Staubli VAL3: ros_server.pjx

--- ros_server.pjx ---
Parameters version=s8.10.3Cs9_BS2093 stackSize=5000 millimeterUnit=true
Program file=dataReceiver.pgx
Program file=dataReceiverIO.pgx
Program file=dataStreamer.pgx
Program file=decodeMsgBody.pgx
Program file=decodeMsgBodyIO.pgx
Program file=decodeMsgHeader.pgx
Program file=decodeMsgHeaderIO.pgx
Program file=decTrajPt.pgx
Program file=decTrajPtFull.pgx
Program file=encodeAck.pgx
Program file=encodeAckIO.pgx
Program file=encodeJState.pgx
Program file=encodeStatus.pgx
Program file=encPrefixHeader.pgx
Program file=encTrajPtAck.pgx
Program file=encTrajPtFAck.pgx
Program file=fetchStatus.pgx
Program file=handleRequest.pgx
Program file=initParams.pgx
Program file=initRosMsg.pgx
Program file=interpolateVel.pgx
Program file=motionControl.pgx
Program file=pushMotion.pgx
Program file=pushMotionIO.pgx
Program file=recvData.pgx
Program file=recvHeartbeat.pgx
Program file=recvMsgBody.pgx
Program file=recvMsgBodyIO.pgx
Program file=recvMsgHeader.pgx
Program file=recvMsgHeaderIO.pgx
Program file=recvRosMsg.pgx
Program file=recvTrajPt.pgx
Program file=recvTrajPtFull.pgx
Program file=screenUpdate.pgx
Program file=sendAck.pgx
Program file=sendAckIO.pgx
Program file=sendData.pgx
Program file=sendRosMsg.pgx
Program file=setupRosMsgs.pgx
Program file=start.pgx
Program file=stop.pgx
Program file=toJointArrayRad.pgx
Program file=toJointRxDeg.pgx
Data file=ros_server.dtx
Library alias=libQueueFuncs path=Disk://ros_libs/QueueFuncs/QueueFuncs.pjx
Library alias=libInterface path=Disk://ros_libs/UserInterface/interfaceDefault/interfaceDefault.pjx autoload=false
Library alias=Staubli path=Disk://ros_libs/Staubli/Staubli.pjx
Library alias=IO path=Disk://ros_libs/IOInterface/IOInterface.pjx
Library alias=SimpleMsg path=Disk://ros_libs/SimpleMessage/SimpleMessage.pjx
Type name=RosSimpleMsg path=Disk://ros_libs/RosSimpleMsg/RosSimpleMsg.pjx
Type name=RobotStatusMsg path=Disk://ros_libs/RobotStatusMsg/RobotStatusMsg.pjx
Type name=JointStateMsg path=Disk://ros_libs/JointStateMsg/JointStateMsg.pjx
Type name=JointTrajPtMsg path=Disk://ros_libs/JointTrajPtMsg/JointTrajPtMsg.pjx
Type name=JointTrajPtFMsg path=Disk://ros_libs/JointTrajPtFMsg/JointTrajPtFMsg.pjx
Type name=JointFbkMsg path=Disk://ros_libs/JointFbkMsg/JointFbkMsg.pjx
Type name=MotionCmd path=Disk://ros_libs/MotionCmd/MotionCmd.pjx
Type name=Header path=Disk://ros_libs/Header/Header.pjx
Type name=Prefix path=Disk://ros_libs/Prefix/Prefix.pjx
Type name=Body path=Disk://ros_libs/Body/Body.pjx
Type name=Queue path=Disk://ros_libs/Queue/Queue.pjx

--- ros_server.dtx ---
public bool bFbkOverrun
public bool bMotionOverrun
public sio siTcpIpFbk = {link=Socket\Feedback}
public sio siTcpIpMotion = {link=Socket\Motion}
public string sStreamTaskName = "publisher"
public string sMotionTaskName
public RosSimpleMsg rosGenericMsg
  [0]
    Header header
      [0]
        num nMsgType
        num nCommType
        num nReplyCode
        num nData[12]
    Prefix prefix
      [0]
        num nLength
        num nData[4]
public tool tTool = {fatherId=flange[0], ioLink=ValveIO\valve1}
public string sTrajPtTaskName
public bool bTrajPtOverrun
public RobotStatusMsg rosStatusMsg
  [0]
    Body body
      [0]
        num nData[28]
    Header header
      [0]
        num nMsgType
        num nCommType
        num nReplyCode
        num nData[12]
    Prefix prefix
      [0]
        num nLength
        num nData[4]
    RobotStatus robotStatus
      [0]
        num nDrivesPowered
        num nEStopped
        num nErrorCode
        num nInError
        num nInMotion
        num nMode
        num nMotionPossible
public JointStateMsg rosJointMsg
  [0]
    Header header
      [0]
        num nMsgType
        num nCommType
        num nReplyCode
        num nData[12]
    Body body
      [0]
        num nData[44]
    JointState jointState
      [0]
        num nSeq
        num nJoints[10]
    Prefix prefix
      [0]
        num nLength
        num nData[4]
public JointTrajPtMsg rosTrajPtMsg
  [0]
    Header header
      [0]
        num nMsgType
        num nCommType
        num nReplyCode
        num nData[12]
    JointTrajPt jointTrajPt
      [0]
        num nSeq
        num nJoints[10]
        num nVelocity
        num nDuration
    Prefix prefix
      [0]
        num nLength
        num nData[4]
    Body body
      [0]
        num nData[52]
public JointTrajPtFMsg rosTrajPtFMsg
  [0]
    Header header
      [0]
        num nMsgType
        num nCommType
        num nReplyCode
        num nData[12]
    Prefix prefix
      [0]
        num nLength
        num nData[4]
    JointTrajPtFull jointTrajPtFull
      [0]
        num nRobotId
        num nSeq
        num nValidFields
        num nTime
        num nPositions[10]
        num nVelocities[10]
        num nAccelerations[10]
    Body body
      [0]
        num nData[136]
public JointFbkMsg rosJointFbkMsg
  [0]
    Header header
      [0]
        num nMsgType
        num nCommType
        num nReplyCode
        num nData[12]
    Prefix prefix
      [0]
        num nLength
        num nData[4]
    JointFeedback jointFeedback
      [0]
        num nRobotId
        num nValidFields
        num nTime
        num nPositions[10]
        num nVelocities[10]
        num nAccelerations[10]
    Body body
      [0]
        num nData[132]
public JointTrajPtFMsg rosTrajPtFAck
  [0]
    Header header
      [0]
        num nMsgType
        num nCommType
        num nReplyCode
        num nData[12]
    Prefix prefix
      [0]
        num nLength
        num nData[4]
    JointTrajPtFull jointTrajPtFull
      [0]
        num nRobotId
        num nSeq
        num nValidFields
        num nTime
        num nPositions[10]
        num nVelocities[10]
        num nAccelerations[10]
    Body body
      [0]
        num nData[136]
public JointTrajPtMsg rosTrajPtAck
  [0]
    Header header
      [0]
        num nMsgType
        num nCommType
        num nReplyCode
        num nData[12]
    JointTrajPt jointTrajPt
      [0]
        num nSeq
        num nJoints[10]
        num nVelocity
        num nDuration
    Prefix prefix
      [0]
        num nLength
        num nData[4]
    Body body
      [0]
        num nData[52]
public bool bScreenOverrun
public string sScreenTaskName
public num nInConnFlag
public num nOutConnFlag
public string sHtbtTaskName
public num nPtsPopped
public bool bStopNow
public num nMotionProgress
public num nMoveId
public num nMovePts
public num nElapsedTime
public num nHeaderTime
public bool bOverwriteVel
public Queue qMoveBuffer
  [0]
    num nPush
    num nPop
    num nElems
    MotionCmd buffer[10]
      [0]
        mdesc mDesc = {leave=0, reach=0}
        num nDuration
        num nSequence
        jointRx jJointRx
      [1]
        mdesc mDesc = {leave=0, reach=0}
        num nDuration
        num nSequence
        jointRx jJointRx
      [2]
        mdesc mDesc = {leave=0, reach=0}
        num nDuration
        num nSequence
        jointRx jJointRx
      [3]
        mdesc mDesc = {leave=0, reach=0}
        num nDuration
        num nSequence
        jointRx jJointRx
      [4]
        mdesc mDesc = {leave=0, reach=0}
        num nDuration
        num nSequence
        jointRx jJointRx
      [5]
        mdesc mDesc = {leave=0, reach=0}
        num nDuration
        num nSequence
        jointRx jJointRx
      [6]
        mdesc mDesc = {leave=0, reach=0}
        num nDuration
        num nSequence
        jointRx jJointRx
      [7]
        mdesc mDesc = {leave=0, reach=0}
        num nDuration
        num nSequence
        jointRx jJointRx
      [8]
        mdesc mDesc = {leave=0, reach=0}
        num nDuration
        num nSequence
        jointRx jJointRx
      [9]
        mdesc mDesc = {leave=0, reach=0}
        num nDuration
        num nSequence
        jointRx jJointRx
public Queue qTrajPtBuffer
  [0]
    num nPush
    num nPop
    num nElems
    MotionCmd buffer[10]
      [0]
        mdesc mDesc = {leave=0, reach=0}
        num nDuration
        num nSequence
        jointRx jJointRx
      [1]
        mdesc mDesc = {leave=0, reach=0}
        num nDuration
        num nSequence
        jointRx jJointRx
      [2]
        mdesc mDesc = {leave=0, reach=0}
        num nDuration
        num nSequence
        jointRx jJointRx
      [3]
        mdesc mDesc = {leave=0, reach=0}
        num nDuration
        num nSequence
        jointRx jJointRx
      [4]
        mdesc mDesc = {leave=0, reach=0}
        num nDuration
        num nSequence
        jointRx jJointRx
      [5]
        mdesc mDesc = {leave=0, reach=0}
        num nDuration
        num nSequence
        jointRx jJointRx
      [6]
        mdesc mDesc = {leave=0, reach=0}
        num nDuration
        num nSequence
        jointRx jJointRx
      [7]
        mdesc mDesc = {leave=0, reach=0}
        num nDuration
        num nSequence
        jointRx jJointRx
      [8]
        mdesc mDesc = {leave=0, reach=0}
        num nDuration
        num nSequence
        jointRx jJointRx
      [9]
        mdesc mDesc = {leave=0, reach=0}
        num nDuration
        num nSequence
        jointRx jJointRx
num nVel[2]
num nStdMsgType{}
  [JOINT_TRAJ_PT] = 11
  [JOINT_TRAJ_PT_FULL] = 14
  [WRITE_SINGLE_IO] = {}
num nCommType{}
  [SERVICE_REQUEST] = 2
mdesc mNomSpeed
num nRecHeader
num nDecHeader = 1
num nRecBody = 2
num nDecBody = 3
num nPushMotion = 4
num nAck = 5
num nReset
public RosSimpleMsg genericIOMsg
  [0]
    Header header
      [0]
        num nMsgType
        num nCommType
        num nReplyCode
        num nData[12]
    Prefix prefix
      [0]
        num nLength
        num nData[4]
num nConnFlagIO
public string sIORequestTaskName
num nConnFlagMotion
public sio siTcpIpIO = {link=Socket\IO}
num ntest
string sTest

--- start.pgx ---
program start()
  local num l_nFbkPeriod
  local num l_nMotionPeriod
  local num l_nTrajPeriod
  local num l_nScreenUpdate
  local string l_sVersionMajor
  local num l_nVersionMajor
  local bool l_bOkMajor
  local string l_sVersionMinor
  local num l_nVersionMinor
  local bool l_bOkMinor
begin
  // Copyright (c) 2016, Ocado Technology - Robotics Research Team
  //
  // Licensed under the Apache License, Version 2.0 (the "License");
  // you may not use this file except in compliance with the License.
  // You may obtain a copy of the License at
  //
  //     http://www.apache.org/licenses/LICENSE-2.0
  //
  // Unless required by applicable law or agreed to in writing, software
  // distributed under the License is distributed on an "AS IS" BASIS,
  // WITHOUT WARRANTIES OR CONDITIONS OF ANY KIND, either express or implied.
  // See the License for the specific language governing permissions and
  // limitations under the License.


  // Load interface library for CS8 or CS9
  //
  // CS9 handles the UI differently than CS8, requires
  // the UI funtions to be loaded in seperate libraries

  if(mid(getVersion("System"),1,1) == "7")
    // CS8 - VAL 3 rev 7
    // Check for VAL 3 version >= 7.7
    l_sVersionMajor = mid(getVersion("VAL3"),1,1)
    l_sVersionMinor = mid(getVersion("VAL3"),2,1)
    toNum(l_sVersionMajor, l_nVersionMajor, l_bOkMajor)
    toNum(l_sVersionMinor, l_nVersionMinor, l_bOkMinor)
    if(!l_bOkMajor or !l_bOkMinor)
      popUpMsg("Error reading VAL 3 version")
      taskKill("ros_server~")
    endIf
    if( !((l_nVersionMajor == 7) and (l_nVersionMinor >= 7)))
      // VAL 3 version is too old
      popUpMsg("Error: VAL 3 version is < 7.7, socket communication will not work!")
      taskKill("ros_server~")
    endIf
    libInterface:libLoad("ros_libs/UserInterface/interfaceCS8")
  elseIf(mid(getVersion("System"),1,1) == "8")
    // CS9 - VAL 3 rev 8
    libInterface:libLoad("ros_libs/UserInterface/interfaceCS9")
  endIf

  // feedback task will run every 20ms (50Hz)
  l_nFbkPeriod=0.02
  //l_nFbkPeriod = 0.032 // 30Hz
  //l_nFbkPeriod = 0.05  // 20Hz
  //l_nFbkPeriod = 1.0   //  1Hz

  // motion control task will run every 4ms (250Hz)
  l_nMotionPeriod = 0.004
  //l_nMotionPeriod=0.012  // 83Hz
  //l_nMotionPeriod = 0.05 // 20Hz

  // data (trajectory) reception task will run every 4ms (250Hz)
  l_nTrajPeriod = 0.004
  // not in use at the moment
  l_nScreenUpdate = 1.0

  sStreamTaskName = "streamerTask"
  sTrajPtTaskName = "trajPtTask"
  sMotionTaskName = "motionTask"
  sIORequestTaskName = "ioRequestTask"
  sScreenTaskName = "screenTask"
  sHtbtTaskName = "htbtTask"

  // initialise TCP/IP parameters
  call initParams()

  // initialise libraries
  call SimpleMsg:init()
  call Staubli:init()
  call IO:init()
  // setup prefix and header of ROS messages
  call setupRosMsgs()

  // socket connection status flags: initially disconnected
  nConnFlagIO = 0
  nInConnFlag = 0
  nOutConnFlag = 0
  nConnFlagMotion = 0

  // flag defining whether velocity to be overwritten to max. vel.
  bOverwriteVel = false

  nPtsPopped = 0
  nMovePts = 0

  // flush buffer of incoming socket
  clearBuffer(siTcpIpIO)
  clearBuffer(siTcpIpMotion)
  // flush buffer of outgoing socket
  clearBuffer(siTcpIpFbk)

  // check if robot is not in emergency stop and wait until estop is reset
  if(esStatus() == 2)
    popUpMsg("Please reset E-Stop")
    wait(esStatus() < 2)
  endIf

  // before anything else, enable power (only works if robot is in remote mode)
  if(!isPowered())
    if(workingMode() >= 4)
      do
        enablePower()
        delay(2)
      until isPowered()
    else
      popUpMsg("Power must be enabled manually")
    endIf
  endIf

  // reset motion, potentially setting a start joint position for calling autoConnect() in the future
  resetMotion()

  // create joint state and robot status streamer task to send data to industrial_robot_client
  taskCreateSync sStreamTaskName, l_nFbkPeriod, bFbkOverrun, dataStreamer()

  // create trajectory point task to receive data from industrial_robot_client
  taskCreateSync sTrajPtTaskName, l_nTrajPeriod, bTrajPtOverrun, dataReceiver()
  //taskCreate sTrajPtTaskName, 100, dataReceiver()

  // create motion task to synchronously apply motion commands to robot
  taskCreateSync sMotionTaskName, l_nMotionPeriod, bMotionOverrun, motionControl()

  // create asynchronous task to handle io requests
  taskCreate sIORequestTaskName, 100, dataReceiverIO(siTcpIpIO, nConnFlagIO, genericIOMsg)

  // create synchronous task to update screen
  //taskCreateSync sScreenTaskName, l_nScreenUpdate, bScreenOverrun, screenUpdate()
  taskCreate sScreenTaskName, 10, screenUpdate()

  // create asynchronous task to receive heartbeat on port 11002
  taskCreate sHtbtTaskName, 10, recvHeartbeat()

end

--- dataReceiver.pgx ---
program dataReceiver()
  local num l_nMsgRecvState
  local num l_nStartTime
begin
  // Copyright (c) 2016, Ocado Technology - Robotics Research Team
  //
  // Licensed under the Apache License, Version 2.0 (the "License");
  // you may not use this file except in compliance with the License.
  // You may obtain a copy of the License at
  //
  //     http://www.apache.org/licenses/LICENSE-2.0
  //
  // Unless required by applicable law or agreed to in writing, software
  // distributed under the License is distributed on an "AS IS" BASIS,
  // WITHOUT WARRANTIES OR CONDITIONS OF ANY KIND, either express or implied.
  // See the License for the specific language governing permissions and
  // limitations under the License.



  // state machine at initial state
  // 0: receive header
  // 1: decode header
  // 2: receive body
  // 3: decode body
  // 4: push motion into buffer
  // 5: send ACK

  // Set variable constants to make sure they were not changed
  nReset=0
  nRecHeader=0
  nDecHeader=1
  nRecBody=2
  nDecBody=3
  nPushMotion=4
  nAck=5

  l_nMsgRecvState=nRecHeader
while (true)
    // usually for state machines a switch-case statement is a neat implementation
    // HOWEVER, at every iteration of while() this task is sequenced and only called
    // after whatever ms is was defined when created.
    // As a result, receiving one single message, pushing motion and sending ACK
    // would take 6 * task period using switch-case statement.
    // The desirable behaviour is to receive and decode a full message, push motion
    // into buffer and then send ACK to client WITHIN ONE ITERATION of while(),
    // hence the if statement sequence below
    l_nStartTime=clock()
    if (l_nMsgRecvState==nRecHeader)
      call recvMsgHeader(l_nMsgRecvState)
    endIf
    nHeaderTime=clock()-l_nStartTime
    if (l_nMsgRecvState==nDecHeader)
      call decodeMsgHeader(l_nMsgRecvState)
    endIf
    if (l_nMsgRecvState==nRecBody)
      call recvMsgBody(l_nMsgRecvState)
    endIf
    if (l_nMsgRecvState==nDecBody)
      call decodeMsgBody(l_nMsgRecvState)
    endIf
    if (l_nMsgRecvState==nPushMotion)
      call pushMotion(l_nMsgRecvState)
    endIf
    if (l_nMsgRecvState==nAck)
      call encodeAck()
      call sendAck(l_nMsgRecvState)
    endIf
    nElapsedTime=clock()-l_nStartTime-nHeaderTime

    // assert state machine is working OK
    if (l_nMsgRecvState<nRecHeader or l_nMsgRecvState>nAck)
      popUpMsg("Data reception state machine error")
    endIf

    // sequence task
    delay(0)


  endWhile
end

--- dataReceiverIO.pgx ---
public program dataReceiverIO(sio& x_sSocket, num& x_nConnFlag, RosSimpleMsg& x_rMsg)
  local num l_nStartTime
  local num l_nMsgRecvState
begin
  // Copyright (c) 2016, Ocado Technology - Robotics Research Team
  //
  // Licensed under the Apache License, Version 2.0 (the "License");
  // you may not use this file except in compliance with the License.
  // You may obtain a copy of the License at
  //
  //     http://www.apache.org/licenses/LICENSE-2.0
  //
  // Unless required by applicable law or agreed to in writing, software
  // distributed under the License is distributed on an "AS IS" BASIS,
  // WITHOUT WARRANTIES OR CONDITIONS OF ANY KIND, either express or implied.
  // See the License for the specific language governing permissions and
  // limitations under the License.



  // state machine at initial state
  // 0: receive header
  // 1: decode header
  // 2: receive body
  // 3: decode body
  // 4: push motion into buffer
  // 5: send ACK

  // Set variable constants to make sure they were not changed
  nReset=0
  nRecHeader=0
  nDecHeader=1
  nRecBody=2
  nDecBody=3
  nPushMotion=4
  nAck=5

  l_nMsgRecvState=nRecHeader

  while(true)
    // usually for state machines a switch-case statement is a neat implementation
    // HOWEVER, at every iteration of while() this task is sequenced and only called
    // after whatever ms is was defined when created.
    // As a result, receiving one single message, pushing motion and sending ACK
    // would take 6 * task period using switch-case statement.
    // The desirable behaviour is to receive and decode a full message, push motion
    // into buffer and then send ACK to client WITHIN ONE ITERATION of while(),
    // hence the if statement sequence below
    l_nStartTime = clock()
    if(l_nMsgRecvState==nRecHeader)
      call recvMsgHeaderIO(x_sSocket, x_nConnFlag, x_rMsg, l_nMsgRecvState)
    endIf

    nHeaderTime = clock() - l_nStartTime
    if(l_nMsgRecvState==nDecHeader)
      call decodeMsgHeaderIO(x_rMsg, l_nMsgRecvState)
      logMsg("Header decoded")
    endIf

    if(l_nMsgRecvState==nRecBody)
      call recvMsgBodyIO(x_sSocket, x_nConnFlag, x_rMsg, l_nMsgRecvState)
      logMsg("Body Recv")
    endIf

    if(l_nMsgRecvState==nDecBody)
      call decodeMsgBodyIO(x_rMsg, l_nMsgRecvState)
      logMsg("Body decoded")
    endIf

    // if(l_nMsgRecvState==nPushMotion)
    //   call pushMotionIO(x_rMsg, l_nMsgRecvState)
    //   logMsg("motion pushed")
    // endIf

     if(l_nMsgRecvState==nPushMotion)
      call handleRequest(x_rMsg, l_nMsgRecvState)
      logMsg("request handled")
    endIf

    if(l_nMsgRecvState==nAck)
      call encodeAckIO(x_rMsg)
      logMsg("Ack encoded")
      call sendAckIO(x_sSocket, x_nConnFlag, x_rMsg, l_nMsgRecvState)
      logMsg("Ack sent")
    endIf
    nElapsedTime = clock() - l_nStartTime - nHeaderTime

    // assert state machine is working OK
    if(l_nMsgRecvState<nRecHeader or l_nMsgRecvState>nAck)
      popUpMsg("Data reception state machine error")
    endIf

    // sequence task
    delay(0)


  endWhile
end

--- dataStreamer.pgx ---
public program dataStreamer()
  local num l_nThrottle
  local jointRx l_jCurrPose
begin
  // Copyright (c) 2016, Ocado Technology - Robotics Research Team
  //
  // Licensed under the Apache License, Version 2.0 (the "License");
  // you may not use this file except in compliance with the License.
  // You may obtain a copy of the License at
  //
  //     http://www.apache.org/licenses/LICENSE-2.0
  //
  // Unless required by applicable law or agreed to in writing, software
  // distributed under the License is distributed on an "AS IS" BASIS,
  // WITHOUT WARRANTIES OR CONDITIONS OF ANY KIND, either express or implied.
  // See the License for the specific language governing permissions and
  // limitations under the License.



  l_nThrottle = 0
  while (true)
    // only attempt to send data if flag indicates that connection is established
    if (nOutConnFlag == 1)
      // fetch current joint positions
      l_jCurrPose=herej()
      // encode and send ROS simple_message ID 10: joint state
      call encodeJState(l_jCurrPose)
      call sendRosMsg(siTcpIpFbk, rosJointMsg.prefix, rosJointMsg.header, rosJointMsg.body, nOutConnFlag)

      // send Robot Status messages 5 times slower than Joint State
      if (l_nThrottle == 5)
        // fetch robot status
        call fetchStatus()
        // encode and send ROS simple_message ID 13: robot status
        call encodeStatus()
        call sendRosMsg(siTcpIpFbk, rosStatusMsg.prefix, rosStatusMsg.header, rosStatusMsg.body, nOutConnFlag)
        l_nThrottle = 0
      endIf
      l_nThrottle = l_nThrottle + 1
    else
      delay(0.1)
    endIf

    // sequence task
    delay(0)
  endWhile
end

--- decodeMsgBody.pgx ---
public program decodeMsgBody(num& x_nMsgRecvState)
  local bool l_bFlag
begin
  // Copyright (c) 2016, Ocado Technology - Robotics Research Team
  //
  // Licensed under the Apache License, Version 2.0 (the "License");
  // you may not use this file except in compliance with the License.
  // You may obtain a copy of the License at
  //
  //     http://www.apache.org/licenses/LICENSE-2.0
  //
  // Unless required by applicable law or agreed to in writing, software
  // distributed under the License is distributed on an "AS IS" BASIS,
  // WITHOUT WARRANTIES OR CONDITIONS OF ANY KIND, either express or implied.
  // See the License for the specific language governing permissions and
  // limitations under the License.



  l_bFlag=false

  switch rosGenericMsg.header.nMsgType
    case nStdMsgType["JOINT_TRAJ_PT"]
      call decTrajPt(l_bFlag)
    break
    case nStdMsgType["JOINT_TRAJ_PT_FULL"]
      call decTrajPtFull(l_bFlag)
    break
    default
    break
  endSwitch

  if (l_bFlag==true)
    // move on to state 4: push motion into buffer
    x_nMsgRecvState=nPushMotion
  else
    // error whilst decoding msg body...
    if (rosGenericMsg.header.nCommType==2)
      switch rosGenericMsg.header.nMsgType
        case nStdMsgType["JOINT_TRAJ_PT"]
          rosTrajPtAck.header.nReplyCode=2
        break
        case nStdMsgType["JOINT_TRAJ_PT_FULL"]
          rosTrajPtFAck.header.nReplyCode=2
        break
        default
        break
      endSwitch
      // jump to state 5: sendAck()
      x_nMsgRecvState=nAck
    else
      // reset state machine, since no ACK is required
      x_nMsgRecvState=nReset
    endIf
  endIf
end

--- decodeMsgBodyIO.pgx ---
public program decodeMsgBodyIO(RosSimpleMsg& x_rMsg, num& x_nMsgRecvState)
  local bool l_bFlag
begin
  // Copyright (c) 2016, Ocado Technology - Robotics Research Team
  //
  // Licensed under the Apache License, Version 2.0 (the "License");
  // you may not use this file except in compliance with the License.
  // You may obtain a copy of the License at
  //
  //     http://www.apache.org/licenses/LICENSE-2.0
  //
  // Unless required by applicable law or agreed to in writing, software
  // distributed under the License is distributed on an "AS IS" BASIS,
  // WITHOUT WARRANTIES OR CONDITIONS OF ANY KIND, either express or implied.
  // See the License for the specific language governing permissions and
  // limitations under the License.



  l_bFlag=false

  //switch x_rMsg.header.nMsgType
  //  case nStdMsgType["JOINT_TRAJ_PT"]
  //    call decTrajPt(l_bFlag)
  //  break
  //  case nStdMsgType["JOINT_TRAJ_PT_FULL"]
  //    call decTrajPtFull(l_bFlag)
  //  break
  //  case Staubli:MsgType.WRITE_SINGLE_IO
      call Staubli:decWriSingIOMsg(l_bFlag)
      logMsg("msgtype")
  //  break
  //  default
  //  break
  //endSwitch

  if (l_bFlag == true)
    // move on to state 4: push motion into buffer
    x_nMsgRecvState=nPushMotion
  else
    // error whilst decoding msg body...
    if (x_rMsg.header.nCommType==2)
      //switch x_rMsg.header.nMsgType
      //  case nStdMsgType["JOINT_TRAJ_PT"]
      //    rosTrajPtAck.header.nReplyCode=2
      //  break
      //  case nStdMsgType["JOINT_TRAJ_PT_FULL"]
      //    rosTrajPtFAck.header.nReplyCode=2
      //  break
      //  case Staubli:MsgType.WRITE_SINGLE_IO
          Staubli:writeSingIOAck.header.nReplyCode=SimpleMsg:ReplyCode.FAILURE
      //  break
      //  default
      //  break
      //endSwitch
      // jump to state 5: sendAck()
      x_nMsgRecvState=nAck
    else
      // reset state machine, since no ACK is required
      x_nMsgRecvState=nReset
    endIf
  endIf
end

--- decodeMsgHeader.pgx ---
public program decodeMsgHeader(num& x_nMsgRecvState)
  local num l_nRetVal
begin
  // Copyright (c) 2016, Ocado Technology - Robotics Research Team
  //
  // Licensed under the Apache License, Version 2.0 (the "License");
  // you may not use this file except in compliance with the License.
  // You may obtain a copy of the License at
  //
  //     http://www.apache.org/licenses/LICENSE-2.0
  //
  // Unless required by applicable law or agreed to in writing, software
  // distributed under the License is distributed on an "AS IS" BASIS,
  // WITHOUT WARRANTIES OR CONDITIONS OF ANY KIND, either express or implied.
  // See the License for the specific language governing permissions and
  // limitations under the License.



  // decode message into generic message first
  l_nRetVal=fromBinary(rosGenericMsg.prefix.nData,4,"-4l",rosGenericMsg.prefix.nLength)
  if (l_nRetVal!=1)
    // error decoding prefix, reset state machine
    x_nMsgRecvState=nReset
    return
  endIf
  l_nRetVal=fromBinary(rosGenericMsg.header.nData,4,"-4l",rosGenericMsg.header.nMsgType)
  if (l_nRetVal!=1)
    // error decoding header (msg type), reset state machine
    x_nMsgRecvState=nReset
    return
  endIf
  l_nRetVal=fromBinary(rosGenericMsg.header.nData[4],4,"-4l",rosGenericMsg.header.nCommType)
  if (l_nRetVal!=1)
    // error decoding header (comm type), reset state machine
    x_nMsgRecvState=nReset
    return
  endIf
  l_nRetVal=fromBinary(rosGenericMsg.header.nData[8],4,"-4l",rosGenericMsg.header.nReplyCode)
  if (l_nRetVal!=1)
    // error decoding header (reply code), reset state machine
    x_nMsgRecvState=nReset
    return
  endIf

  // no errors detected whilst decoding prefix and header
  // move on to state 2: receive msg body
  x_nMsgRecvState=nRecBody
end

--- decodeMsgHeaderIO.pgx ---
public program decodeMsgHeaderIO(RosSimpleMsg& x_rMsg, num& x_nMsgRecvState)
  local num l_nRetVal
begin
  // Copyright (c) 2016, Ocado Technology - Robotics Research Team
  //
  // Licensed under the Apache License, Version 2.0 (the "License");
  // you may not use this file except in compliance with the License.
  // You may obtain a copy of the License at
  //
  //     http://www.apache.org/licenses/LICENSE-2.0
  //
  // Unless required by applicable law or agreed to in writing, software
  // distributed under the License is distributed on an "AS IS" BASIS,
  // WITHOUT WARRANTIES OR CONDITIONS OF ANY KIND, either express or implied.
  // See the License for the specific language governing permissions and
  // limitations under the License.



  // decode message into generic message first
  l_nRetVal=fromBinary(x_rMsg.prefix.nData,4,"-4l",x_rMsg.prefix.nLength)
  if (l_nRetVal!=1)
    // error decoding prefix, reset state machine
    x_nMsgRecvState=nReset
    return
  endIf
  l_nRetVal=fromBinary(x_rMsg.header.nData,4,"-4l",x_rMsg.header.nMsgType)
  if (l_nRetVal!=1)
    // error decoding header (msg type), reset state machine
    x_nMsgRecvState=nReset
    return
  endIf
  l_nRetVal=fromBinary(x_rMsg.header.nData[4],4,"-4l",x_rMsg.header.nCommType)
  if (l_nRetVal!=1)
    // error decoding header (comm type), reset state machine
    x_nMsgRecvState=nReset
    return
  endIf
  l_nRetVal=fromBinary(x_rMsg.header.nData[8],4,"-4l",x_rMsg.header.nReplyCode)
  if (l_nRetVal!=1)
    // error decoding header (reply code), reset state machine
    x_nMsgRecvState=nReset
    return
  endIf

  // no errors detected whilst decoding prefix and header
  // move on to state 2: receive msg body
  x_nMsgRecvState=nRecBody
end

--- encodeAck.pgx ---
public program encodeAck()
begin
  // Copyright (c) 2016, Ocado Technology - Robotics Research Team
  //
  // Licensed under the Apache License, Version 2.0 (the "License");
  // you may not use this file except in compliance with the License.
  // You may obtain a copy of the License at
  //
  //     http://www.apache.org/licenses/LICENSE-2.0
  //
  // Unless required by applicable law or agreed to in writing, software
  // distributed under the License is distributed on an "AS IS" BASIS,
  // WITHOUT WARRANTIES OR CONDITIONS OF ANY KIND, either express or implied.
  // See the License for the specific language governing permissions and
  // limitations under the License.



  switch rosGenericMsg.header.nMsgType
    case nStdMsgType["JOINT_TRAJ_PT"]
      call encTrajPtAck()
    break
    case nStdMsgType["JOINT_TRAJ_PT_FULL"]
      call encTrajPtFAck()
    break
    default
    break
  endSwitch
end

--- encodeAckIO.pgx ---
public program encodeAckIO(RosSimpleMsg& x_rMsg)
begin
  // Copyright (c) 2016, Ocado Technology - Robotics Research Team
  //
  // Licensed under the Apache License, Version 2.0 (the "License");
  // you may not use this file except in compliance with the License.
  // You may obtain a copy of the License at
  //
  //     http://www.apache.org/licenses/LICENSE-2.0
  //
  // Unless required by applicable law or agreed to in writing, software
  // distributed under the License is distributed on an "AS IS" BASIS,
  // WITHOUT WARRANTIES OR CONDITIONS OF ANY KIND, either express or implied.
  // See the License for the specific language governing permissions and
  // limitations under the License.



  switch x_rMsg.header.nMsgType
    case nStdMsgType["JOINT_TRAJ_PT"]
      call encTrajPtAck()
    break
    case nStdMsgType["JOINT_TRAJ_PT_FULL"]
      call encTrajPtFAck()
    break

    //Staubli specific
    case Staubli:MsgType.WRITE_SINGLE_IO
      call Staubli:encWriSingIOAck()
    break
    default
    break
  endSwitch
end

--- handleRequest.pgx ---
public program handleRequest(RosSimpleMsg& x_rMsg, num& x_nMsgRecvState)
  local bool l_bOk
  local num l_nModuleId
  local num l_nPin
  local bool l_bState
begin
  // Copyright (c) 2021, Institute for Factory Automation and Production Systems (FAPS)
  //
  // Licensed under the Apache License, Version 2.0 (the "License");
  // you may not use this file except in compliance with the License.
  // You may obtain a copy of the License at
  //
  //     http://www.apache.org/licenses/LICENSE-2.0
  //
  // Unless required by applicable law or agreed to in writing, software
  // distributed under the License is distributed on an "AS IS" BASIS,
  // WITHOUT WARRANTIES OR CONDITIONS OF ANY KIND, either express or implied.
  // See the License for the specific language governing permissions and
  // limitations under the License.


  // assume success to push motion
  l_bOk=true

  // handle request
  // switch x_rMsg.header.nMsgType
    // case Staubli:MsgType.SET_DRIVE_POWER
    //   if (Staubli:setDrvPwrMsg.bDrivePower==true and isPowered()==false)
    //     enablePower()
    //   elseIf (Staubli:setDrvPwrMsg.bDrivePower==false and isPowered()==true)
    //     disablePower()
    //   else
        // nothing to do
    //   endIf
    // break
    // case Staubli:MsgType.WRITE_SINGLE_IO
      l_nModuleId=Staubli:writeSingIOMsg.writeSingleIO.nModuleId
      l_nPin=Staubli:writeSingIOMsg.writeSingleIO.nPin
      l_bState=Staubli:writeSingIOMsg.writeSingleIO.bState
      call IO:writeSingle(l_nModuleId,l_nPin,l_bState,l_bOk)
    // break
    // unknown message type
    // default
    //   l_bOk=false
    // break
  // endSwitch

  //region @check_success -- check whether handling request was successful
  if (l_bOk)
  else
    // could not handle request
    // thus ACK should flag FAILURE, but only if comm type is request
    if (x_rMsg.header.nCommType==SimpleMsg:CommType.SERVICE_REQUEST)
      // switch x_rMsg.header.nMsgType
      //  case Staubli:MsgType.SET_DRIVE_POWER
      //    Staubli:setDrvPwrAck.header.nReplyCode=SimpleMsg:ReplyCode.FAILURE
      //  break
      //  case Staubli:MsgType.WRITE_SINGLE_IO
          Staubli:writeSingIOAck.header.nReplyCode=SimpleMsg:ReplyCode.FAILURE
      //  break
      //  default
      //  break
      //endSwitch
    endIf
  endIf
  //endregion

  //region @check_reply -- check whether service reply (ACK) should be sent
  if (x_rMsg.header.nCommType==SimpleMsg:CommType.SERVICE_REQUEST)
    // comm type request requires ACK
    // x_nMsgRecvState = MsgRecvState.SEND_ACK
    x_nMsgRecvState = nAck
  else
    // other comm types (e.g., topic) does not require ACK, hence skip state
    // x_nMsgRecvState = MsgRecvState.RECEIVE_HEADER
    x_nMsgRecvState = nRecHeader
  endIf
  //endregion
end

--- initParams.pgx ---
public program initParams()
  local num l_nRetVal
begin
  // Copyright (c) 2016, Ocado Technology - Robotics Research Team
  //
  // Licensed under the Apache License, Version 2.0 (the "License");
  // you may not use this file except in compliance with the License.
  // You may obtain a copy of the License at
  //
  //     http://www.apache.org/licenses/LICENSE-2.0
  //
  // Unless required by applicable law or agreed to in writing, software
  // distributed under the License is distributed on an "AS IS" BASIS,
  // WITHOUT WARRANTIES OR CONDITIONS OF ANY KIND, either express or implied.
  // See the License for the specific language governing permissions and
  // limitations under the License.



  l_nRetVal=sioCtrl(siTcpIpMotion,"timeout",-1)
  if(l_nRetVal!=0)
    popUpMsg("Error while setting consumer timeout")
  endIf

  l_nRetVal=sioCtrl(siTcpIpFbk,"timeout",-1)
  if(l_nRetVal!=0)
    popUpMsg("Error while setting producer timeout")
  endIf

  l_nRetVal=sioCtrl(siTcpIpIO, "timeout", -1)
  if(l_nRetVal!=0)
    popUpMsg("Error while setting IO timeout")
  endIf
end

--- initRosMsg.pgx ---
public program initRosMsg()
begin
  // Copyright (c) 2016, Ocado Technology - Robotics Research Team
  //
  // Licensed under the Apache License, Version 2.0 (the "License");
  // you may not use this file except in compliance with the License.
  // You may obtain a copy of the License at
  //
  //     http://www.apache.org/licenses/LICENSE-2.0
  //
  // Unless required by applicable law or agreed to in writing, software
  // distributed under the License is distributed on an "AS IS" BASIS,
  // WITHOUT WARRANTIES OR CONDITIONS OF ANY KIND, either express or implied.
  // See the License for the specific language governing permissions and
  // limitations under the License.



  // Joint state message (ID 10)
  // prefix length = 12 + 44
  rosJointMsg.prefix.nLength=56
  rosJointMsg.header.nMsgType=10
  rosJointMsg.header.nCommType=1
  rosJointMsg.header.nReplyCode=0
  // sequence
  rosJointMsg.jointState.nSeq=0



  // Trajectory point message (ID 11)
  // prefix length = 12 + 52
  rosTrajPtAck.prefix.nLength=64
  rosTrajPtAck.header.nMsgType=11
  rosTrajPtAck.header.nCommType=3
  // reply: 1 = success, 2 = failure
  rosTrajPtAck.header.nReplyCode=1
  // joints are assumed to be initiliased to zero

  // the message bellow will be filled upon reception
  rosTrajPtMsg.prefix.nLength=64



  // Robot status message (ID 13)
  // prefix length = 12 + 28
  rosStatusMsg.prefix.nLength=40
  rosStatusMsg.header.nMsgType=13
  rosStatusMsg.header.nCommType=1
  rosStatusMsg.header.nReplyCode=0

  // Trajectory point full message (ID 14)
  // prefix length = 12 + 136
  rosTrajPtFAck.prefix.nLength=148
  rosTrajPtFAck.header.nMsgType=14
  rosTrajPtFAck.header.nCommType=3
  // reply: 1 = success, 2 = failure
  rosTrajPtFAck.header.nReplyCode=1
  // body (data) assumed to be initialised to zero

  // the message bellow will be filled upon reception
  rosTrajPtFMsg.prefix.nLength=148



  // Joint feedback message (ID 15)
  // prefix length = 12 + 132
  rosJointFbkMsg.prefix.nLength=144
  rosJointFbkMsg.header.nMsgType=15
  rosJointFbkMsg.header.nCommType=1
  rosJointFbkMsg.header.nReplyCode=0
end

--- pushMotion.pgx ---
public program pushMotion(num& x_nMsgRecvState)
  local bool l_bOk
  local MotionCmd l_mTrajPt
  local num l_nCounter
  local num l_nJointError
begin
  // Copyright (c) 2016, Ocado Technology - Robotics Research Team
  //
  // Licensed under the Apache License, Version 2.0 (the "License");
  // you may not use this file except in compliance with the License.
  // You may obtain a copy of the License at
  //
  //     http://www.apache.org/licenses/LICENSE-2.0
  //
  // Unless required by applicable law or agreed to in writing, software
  // distributed under the License is distributed on an "AS IS" BASIS,
  // WITHOUT WARRANTIES OR CONDITIONS OF ANY KIND, either express or implied.
  // See the License for the specific language governing permissions and
  // limitations under the License.



  switch rosGenericMsg.header.nMsgType
    case nStdMsgType["JOINT_TRAJ_PT"]
      l_mTrajPt.nSequence=rosTrajPtMsg.jointTrajPt.nSeq

      // ROS joint position values are in rad, but VAL3 uses degrees
      call toJointRxDeg(rosTrajPtMsg.jointTrajPt.nJoints,l_mTrajPt.jJointRx)

      // from industrial_robot_client/src/joint_trajectory_interface.cpp
      // JointTrajectoryInterface::trajectory_to_msgs()
      // JointTrajectoryInterface::calc_speed()
      // velocity is converted to a scalar value representing % of max velocity,
      // such that 0.2 = 20% of maximum joint speed
      l_mTrajPt.mDesc.vel=limit((rosTrajPtMsg.jointTrajPt.nVelocity*100),0,100)
      l_mTrajPt.nDuration=rosTrajPtMsg.jointTrajPt.nDuration

    break
    case nStdMsgType["JOINT_TRAJ_PT_FULL"]
      l_mTrajPt.nSequence=rosTrajPtFMsg.jointTrajPtFull.nSeq
      l_mTrajPt.nDuration=rosTrajPtFMsg.jointTrajPtFull.nTime

      // ROS joint position values are in rad, but VAL3 uses degrees
      call toJointRxDeg(rosTrajPtFMsg.jointTrajPtFull.nPositions,l_mTrajPt.jJointRx)

      // from industrial_robot_client/src/joint_trajectory_interface.cpp
      // JointTrajectoryInterface::trajectory_to_msgs()
      // JointTrajectoryInterface::calc_speed()
      // velocity is converted to a scalar value representing % of max velocity,
      // such that 0.2 = 20% of maximum joint speed
      l_mTrajPt.mDesc.vel=limit((rosTrajPtFMsg.jointTrajPtFull.nVelocities[0]*100),0,100)
      // not sure about accelerations as yet
      l_mTrajPt.mDesc.accel=rosTrajPtFMsg.jointTrajPtFull.nAccelerations[0]
      l_mTrajPt.mDesc.decel=l_mTrajPt.mDesc.accel
    break
    default
    break
  endSwitch

  // see github.com/ros-industrial/industrial_core/simple_message/include/simple_message/joint_traj_pt.h
  if (l_mTrajPt.nSequence==-4)
    // set flag to stop immediately
    bStopNow=true
  else
    // check whether velocity value should be overwritten with value set on teach pendant
    if (bOverwriteVel==true)
      // overwrite velocity (and acceleration - ?)
      //l_mTrajPt.mDesc.vel = getMonitorSpeed()
      // explicitly setting accel and decel to VAL3 default values
      l_mTrajPt.mDesc.accel=mNomSpeed.accel
      l_mTrajPt.mDesc.decel=mNomSpeed.decel
    endIf
    // only push motion into buffer if not a STOP message
    // and if joint positions are within software joint limits
    // and if velocity is greater than zero (beucase movej() will not accept vel <= 0)
    if (isInRange(l_mTrajPt.jJointRx) and l_mTrajPt.mDesc.vel>0)
      call libQueueFuncs:push(qTrajPtBuffer,l_mTrajPt,l_bOk)
    else
      l_bOk=false
    endIf

    if (l_bOk==false)
      // could not push trajectory point into buffer
      // thus ACK should flag FAILURE, but only if comm type is request
      if (rosGenericMsg.header.nCommType==nCommType["SERVICE_REQUEST"])
        switch rosGenericMsg.header.nMsgType
          case nStdMsgType["JOINT_TRAJ_PT"]
            rosTrajPtAck.header.nReplyCode=2
          break
          case nStdMsgType["JOINT_TRAJ_PT_FULL"]
            rosTrajPtFAck.header.nReplyCode=2
          break
          default
          break
        endSwitch
      endIf
    endIf
  endIf
  // check whether ACK should be sent
  if (rosGenericMsg.header.nCommType==nCommType["SERVICE_REQUEST"])
    // comm type request requires ACK
    x_nMsgRecvState=nAck
  else
    // other comm types (e.g., topic) does not require ACK, hence skip state
    x_nMsgRecvState=nReset
  endIf
end

--- pushMotionIO.pgx ---
public program pushMotionIO(RosSimpleMsg& x_rMsg, num& x_nMsgRecvState)
  local bool l_bOk
  local num l_nCounter
  local num l_nJointError
  local MotionCmd l_mTrajPt
begin
  // Copyright (c) 2016, Ocado Technology - Robotics Research Team
  //
  // Licensed under the Apache License, Version 2.0 (the "License");
  // you may not use this file except in compliance with the License.
  // You may obtain a copy of the License at
  //
  //     http://www.apache.org/licenses/LICENSE-2.0
  //
  // Unless required by applicable law or agreed to in writing, software
  // distributed under the License is distributed on an "AS IS" BASIS,
  // WITHOUT WARRANTIES OR CONDITIONS OF ANY KIND, either express or implied.
  // See the License for the specific language governing permissions and
  // limitations under the License.



  switch x_rMsg.header.nMsgType
    case nStdMsgType["JOINT_TRAJ_PT"]
      l_mTrajPt.nSequence=rosTrajPtMsg.jointTrajPt.nSeq

      // ROS joint position values are in rad, but VAL3 uses degrees
      call toJointRxDeg(rosTrajPtMsg.jointTrajPt.nJoints, l_mTrajPt.jJointRx)

      // from industrial_robot_client/src/joint_trajectory_interface.cpp
      // JointTrajectoryInterface::trajectory_to_msgs()
      // JointTrajectoryInterface::calc_speed()
      // velocity is converted to a scalar value representing % of max velocity,
      // such that 0.2 = 20% of maximum joint speed
      l_mTrajPt.mDesc.vel= limit((rosTrajPtMsg.jointTrajPt.nVelocity * 100), 0, 100)
      l_mTrajPt.nDuration=rosTrajPtMsg.jointTrajPt.nDuration

    break
    case nStdMsgType["JOINT_TRAJ_PT_FULL"]
      l_mTrajPt.nSequence=rosTrajPtFMsg.jointTrajPtFull.nSeq
      l_mTrajPt.nDuration=rosTrajPtFMsg.jointTrajPtFull.nTime

      // ROS joint position values are in rad, but VAL3 uses degrees
      call toJointRxDeg(rosTrajPtFMsg.jointTrajPtFull.nPositions, l_mTrajPt.jJointRx)

      // from industrial_robot_client/src/joint_trajectory_interface.cpp
      // JointTrajectoryInterface::trajectory_to_msgs()
      // JointTrajectoryInterface::calc_speed()
      // velocity is converted to a scalar value representing % of max velocity,
      // such that 0.2 = 20% of maximum joint speed
      l_mTrajPt.mDesc.vel= limit((rosTrajPtFMsg.jointTrajPtFull.nVelocities[0] * 100), 0, 100)
      // not sure about accelerations as yet
      l_mTrajPt.mDesc.accel=rosTrajPtFMsg.jointTrajPtFull.nAccelerations[0]
      l_mTrajPt.mDesc.decel=l_mTrajPt.mDesc.accel
    break
    default
    break
  endSwitch

  // see github.com/ros-industrial/industrial_core/simple_message/include/simple_message/joint_traj_pt.h
  if(l_mTrajPt.nSequence==-4)
    // set flag to stop immediately
    bStopNow=true
  else
    // check whether velocity value should be overwritten with value set on teach pendant
    if(bOverwriteVel == true)
      // overwrite velocity (and acceleration - ?)
      //l_mTrajPt.mDesc.vel = getMonitorSpeed()
      // explicitly setting accel and decel to VAL3 default values
      l_mTrajPt.mDesc.accel = mNomSpeed.accel
      l_mTrajPt.mDesc.decel = mNomSpeed.decel
    endIf
    // only push motion into buffer if not a STOP message
    // and if joint positions are within software joint limits
    // and if velocity is greater than zero (beucase movej() will not accept vel <= 0)
    if(isInRange(l_mTrajPt.jJointRx) and l_mTrajPt.mDesc.vel > 0)
      call libQueueFuncs:push(qTrajPtBuffer,l_mTrajPt,l_bOk)
    else
      l_bOk = false
    endIf

    if(l_bOk==false)
      // could not push trajectory point into buffer
      // thus ACK should flag FAILURE, but only if comm type is request
      if(x_rMsg.header.nCommType==nCommType["SERVICE_REQUEST"])
        switch x_rMsg.header.nMsgType
          case nStdMsgType["JOINT_TRAJ_PT"]
            rosTrajPtAck.header.nReplyCode=2
          break
          case nStdMsgType["JOINT_TRAJ_PT_FULL"]
            rosTrajPtFAck.header.nReplyCode=2
          break
          default
          break
        endSwitch
      endIf
    endIf
  endIf
  // check whether ACK should be sent
  if(x_rMsg.header.nCommType == nCommType["SERVICE_REQUEST"])
    // comm type request requires ACK
    x_nMsgRecvState = nAck
  else
    // other comm types (e.g., topic) does not require ACK, hence skip state
    x_nMsgRecvState = nReset
  endIf
end

--- recvMsgBody.pgx ---
public program recvMsgBody(num& x_nMsgRecvState)
  local bool l_bFlag
begin
  // Copyright (c) 2016, Ocado Technology - Robotics Research Team
  //
  // Licensed under the Apache License, Version 2.0 (the "License");
  // you may not use this file except in compliance with the License.
  // You may obtain a copy of the License at
  //
  //     http://www.apache.org/licenses/LICENSE-2.0
  //
  // Unless required by applicable law or agreed to in writing, software
  // distributed under the License is distributed on an "AS IS" BASIS,
  // WITHOUT WARRANTIES OR CONDITIONS OF ANY KIND, either express or implied.
  // See the License for the specific language governing permissions and
  // limitations under the License.



  l_bFlag=false

  switch rosGenericMsg.header.nMsgType
    case nStdMsgType["JOINT_TRAJ_PT"]
      call recvTrajPt(l_bFlag)
    break
    case nStdMsgType["JOINT_TRAJ_PT_FULL"]
      call recvTrajPtFull(l_bFlag)
    break
    default
    break
  endSwitch

  if (l_bFlag==true)
    // move on to state 3: decode msg body
    x_nMsgRecvState=nDecBody
  else
    // error whilst receiving msg body, reset state machine
    x_nMsgRecvState=nReset
  endIf
end

--- recvMsgBodyIO.pgx ---
public program recvMsgBodyIO(sio& x_sSocket, num& x_nConnFlag, RosSimpleMsg& x_rMsg, num& x_nMsgRecvState)
  local bool l_bFlag
begin
  // Copyright (c) 2016, Ocado Technology - Robotics Research Team
  //
  // Licensed under the Apache License, Version 2.0 (the "License");
  // you may not use this file except in compliance with the License.
  // You may obtain a copy of the License at
  //
  //     http://www.apache.org/licenses/LICENSE-2.0
  //
  // Unless required by applicable law or agreed to in writing, software
  // distributed under the License is distributed on an "AS IS" BASIS,
  // WITHOUT WARRANTIES OR CONDITIONS OF ANY KIND, either express or implied.
  // See the License for the specific language governing permissions and
  // limitations under the License.

  logMsg("message")
      logMsg(toString("", x_rMsg.header.nData[0]))
      logMsg(toString("", x_rMsg.header.nData[1]))
      logMsg(toString("", x_rMsg.header.nData[2]))
      logMsg(toString("", x_rMsg.header.nData[3]))
      logMsg(toString("", x_rMsg.header.nData[4]))
      logMsg(toString("", x_rMsg.header.nData[5]))
      logMsg(toString("", x_rMsg.header.nData[6]))
      logMsg(toString("", x_rMsg.header.nData[7]))
      logMsg(toString("", x_rMsg.header.nData[8]))
      logMsg(toString("", x_rMsg.header.nData[9]))
      logMsg(toString("", x_rMsg.header.nData[10]))
      logMsg(toString("", x_rMsg.header.nData[11]))
      logMsg("prefix")
      logMsg(toString("", x_rMsg.prefix.nData[0]))
      logMsg(toString("", x_rMsg.prefix.nData[1]))
      logMsg(toString("", x_rMsg.prefix.nData[2]))
      logMsg(toString("", x_rMsg.prefix.nData[3]))


  l_bFlag=false
  ntest = x_rMsg.header.nMsgType
  sTest = toString("", ntest)
  //logMsg(stest)
  //switch x_rMsg.header.nMsgType
  //  case nStdMsgType["JOINT_TRAJ_PT"]
  //    call recvTrajPt(l_bFlag)
  //  break
  //  case nStdMsgType["JOINT_TRAJ_PT_FULL"]
  //    call recvTrajPtFull(l_bFlag)
  //  break
  //  case Staubli:MsgType.WRITE_SINGLE_IO
      call recvRosMsg (x_sSocket,Staubli:writeSingIOMsg.prefix,Staubli:writeSingIOMsg.header,Staubli:writeSingIOMsg.body,x_nConnFlag, x_rMsg, l_bFlag)
  //  break
  //  default
  //  break
  //endSwitch

  if (l_bFlag == true)
    // move on to state 3: decode msg body
    x_nMsgRecvState=nDecBody
  else
    // error whilst receiving msg body, reset state machine
    x_nMsgRecvState=nReset
  endIf
end

--- recvMsgHeader.pgx ---
public program recvMsgHeader(num& x_nMsgRecvState)
  local bool l_bFlag
begin
  // Copyright (c) 2016, Ocado Technology - Robotics Research Team
  //
  // Licensed under the Apache License, Version 2.0 (the "License");
  // you may not use this file except in compliance with the License.
  // You may obtain a copy of the License at
  //
  //     http://www.apache.org/licenses/LICENSE-2.0
  //
  // Unless required by applicable law or agreed to in writing, software
  // distributed under the License is distributed on an "AS IS" BASIS,
  // WITHOUT WARRANTIES OR CONDITIONS OF ANY KIND, either express or implied.
  // See the License for the specific language governing permissions and
  // limitations under the License.



  // attempt to receive message prefix and header
  call recvData(siTcpIpMotion,rosGenericMsg.prefix.nData,nInConnFlag,l_bFlag)
  if (l_bFlag==true)
    call recvData(siTcpIpMotion,rosGenericMsg.header.nData,nInConnFlag,l_bFlag)
  endIf

  if (l_bFlag==true)
    // move on to state 1: decode header
    x_nMsgRecvState=nDecHeader
  else
    // error: reset state to 0: receive header
    x_nMsgRecvState=nReset
  endIf
end

--- recvMsgHeaderIO.pgx ---
public program recvMsgHeaderIO(sio& x_sSocket, num& x_nConnFlag, RosSimpleMsg& x_rMsg, num& x_nMsgRecvState)
  local bool l_bFlag
begin
  // Copyright (c) 2016, Ocado Technology - Robotics Research Team
  //
  // Licensed under the Apache License, Version 2.0 (the "License");
  // you may not use this file except in compliance with the License.
  // You may obtain a copy of the License at
  //
  //     http://www.apache.org/licenses/LICENSE-2.0
  //
  // Unless required by applicable law or agreed to in writing, software
  // distributed under the License is distributed on an "AS IS" BASIS,
  // WITHOUT WARRANTIES OR CONDITIONS OF ANY KIND, either express or implied.
  // See the License for the specific language governing permissions and
  // limitations under the License.



  // attempt to receive message prefix and header
  call recvData(x_sSocket,x_rMsg.prefix.nData,x_nConnFlag,l_bFlag)
  if (l_bFlag == true)
    call recvData(x_sSocket,x_rMsg.header.nData,x_nConnFlag,l_bFlag)
  endIf

  if (l_bFlag == true)
    // move on to state 1: decode header
    x_nMsgRecvState=nDecHeader
  else
    // error: reset state to 0: receive header
    x_nMsgRecvState=nReset
  endIf
end

--- recvRosMsg.pgx ---
program recvRosMsg(sio& x_sSocket, Prefix& x_pPrefix, Header& x_hHeader, Body& x_bBody, num& x_nConnFlag, RosSimpleMsg& x_rMsg, bool& x_bValidFlag)
begin
  // Copyright (c) 2021, Institute for Factory Automation and Production Systems (FAPS)
  //
  // Licensed under the Apache License, Version 2.0 (the "License");
  // you may not use this file except in compliance with the License.
  // You may obtain a copy of the License at
  //
  //     http://www.apache.org/licenses/LICENSE-2.0
  //
  // Unless required by applicable law or agreed to in writing, software
  // distributed under the License is distributed on an "AS IS" BASIS,
  // WITHOUT WARRANTIES OR CONDITIONS OF ANY KIND, either express or implied.
  // See the License for the specific language governing permissions and
  // limitations under the License.


  // attempt to receive the data of the message (prefix and header are in x_msg)
  x_pPrefix.nLength=x_rMsg.prefix.nLength
  x_hHeader.nMsgType=x_rMsg.header.nMsgType
  x_hHeader.nCommType=x_rMsg.header.nCommType
  x_hHeader.nReplyCode=x_rMsg.header.nReplyCode

  call recvData(x_sSocket,x_bBody.nData,x_nConnFlag,x_bValidFlag)
end

--- sendAck.pgx ---
public program sendAck(num& x_nMsgRecvState)
begin
  // Copyright (c) 2016, Ocado Technology - Robotics Research Team
  //
  // Licensed under the Apache License, Version 2.0 (the "License");
  // you may not use this file except in compliance with the License.
  // You may obtain a copy of the License at
  //
  //     http://www.apache.org/licenses/LICENSE-2.0
  //
  // Unless required by applicable law or agreed to in writing, software
  // distributed under the License is distributed on an "AS IS" BASIS,
  // WITHOUT WARRANTIES OR CONDITIONS OF ANY KIND, either express or implied.
  // See the License for the specific language governing permissions and
  // limitations under the License.



  switch rosGenericMsg.header.nMsgType
    case nStdMsgType["JOINT_TRAJ_PT"]
      call sendRosMsg(siTcpIpMotion,rosTrajPtAck.prefix,rosTrajPtAck.header,rosTrajPtAck.body,nInConnFlag)
    break
    case nStdMsgType["JOINT_TRAJ_PT_FULL"]
      call sendRosMsg(siTcpIpMotion,rosTrajPtFAck.prefix,rosTrajPtFAck.header,rosTrajPtFAck.body,nInConnFlag)
    break
    default
    break
  endSwitch

  // regardless of result from sending ACK
  // reset state machine to receive new messages
  x_nMsgRecvState=nReset
end

--- sendAckIO.pgx ---
public program sendAckIO(sio& x_sSocket, num& x_nConnFlag, RosSimpleMsg& x_rMsg, num& x_nMsgRecvState)
begin
  // Copyright (c) 2016, Ocado Technology - Robotics Research Team
  //
  // Licensed under the Apache License, Version 2.0 (the "License");
  // you may not use this file except in compliance with the License.
  // You may obtain a copy of the License at
  //
  //     http://www.apache.org/licenses/LICENSE-2.0
  //
  // Unless required by applicable law or agreed to in writing, software
  // distributed under the License is distributed on an "AS IS" BASIS,
  // WITHOUT WARRANTIES OR CONDITIONS OF ANY KIND, either express or implied.
  // See the License for the specific language governing permissions and
  // limitations under the License.



  switch x_rMsg.header.nMsgType
    case nStdMsgType["JOINT_TRAJ_PT"]
      call sendRosMsg(siTcpIpMotion, rosTrajPtAck.prefix, rosTrajPtAck.header, rosTrajPtAck.body, nInConnFlag)
    break
    case nStdMsgType["JOINT_TRAJ_PT_FULL"]
      call sendRosMsg(siTcpIpMotion, rosTrajPtFAck.prefix, rosTrajPtFAck.header, rosTrajPtFAck.body, nInConnFlag)
    break
    case Staubli:MsgType.WRITE_SINGLE_IO
      call sendRosMsg(x_sSocket, Staubli:writeSingIOAck.prefix, Staubli:writeSingIOAck.header, Staubli:writeSingIOAck.body, x_nConnFlag)
    break
    default
    break
  endSwitch

  // regardless of result from sending ACK
  // reset state machine to receive new messages
  x_nMsgRecvState=nReset
end
